FUNCTION_BLOCK ALI_AUI_DEMUX_5 (* ALI demultiplexor (generic FB) Adapter-Ausgang wird nur bei Wertänderung aktualisiert (Event nur bei tatsächlicher Änderung). *)
  (* Standard: 61499-2; Description: Copyright (c) 2026 HR Agrartechnik GmbH This program and the accompanying materials are made available under the terms of the Eclipse Public License 2.0 which is available at https://www.eclipse.org/legal/epl-2.0/ SPDX-License-Identifier: EPL-2.0 *)
  (* Version 1.0, 2026-08-13, Franz Höpfinger, HR Agrartechnik GmbH *)
  PACKAGE adapter::selection::unidirectional;
  {SET_ATTRIBUTE(eclipse4diac::core::GenericClassName, 'GEN_ALI_AUI_DEMUX')}
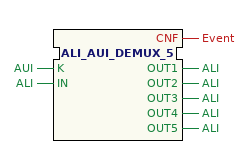
  EVENT_OUTPUT
    CNF; (* Confirmation of Set Index K *)
  END_EVENT
  SOCKETS
    K : adapter::types::unidirectional::AUI; (* index *)
    IN : adapter::types::unidirectional::ALI; (* Input Value to demultiplex *)
  END_SOCKETS
  PLUGS
    OUT1 : adapter::types::unidirectional::ALI; (* Output value 1 (selected when K = 0) *)
    OUT2 : adapter::types::unidirectional::ALI; (* Output value 2 (selected when K = 1) *)
    OUT3 : adapter::types::unidirectional::ALI; (* Output value 3 (selected when K = 2) *)
    OUT4 : adapter::types::unidirectional::ALI; (* Output value 4 (selected when K = 3) *)
    OUT5 : adapter::types::unidirectional::ALI; (* Output value 5 (selected when K = 4) *)
  END_PLUGS
END_FUNCTION_BLOCK
